(* IEC 61131-3 sources: AXOpen/src/components.robotics/ctrl/test, 2 files *)

(* ---- CylinderTests.st ---- *)
USING AXOpen.Components.Robotics;
USING AXOpen.Core;
USING AXOpen.Rtc;
USING AXOpen.Logging;

NAMESPACE Cylinder.Tests
    {S7.extern=ReadWrite}
    CLASS TestContext IMPLEMENTS AXOpen.Core.IAxoContext
        VAR
            _openCounter : ULINT;
            _closeCounter : ULINT;
        END_VAR

        METHOD PUBLIC Open : ULINT
            _openCounter := _openCounter + ULINT#1;
        END_METHOD

        METHOD PUBLIC Close : ULINT
            _closeCounter := _closeCounter + ULINT#1;
        END_METHOD

        METHOD PUBLIC CreateIdentity : ULINT
            ;
        END_METHOD

        METHOD PUBLIC OpenCycleCount : ULINT
            OpenCycleCount := _openCounter;
        END_METHOD

        METHOD PUBLIC GetRtc : AXOpen.Rtc.IAxoRtc
            ;
        END_METHOD

        METHOD PUBLIC InjectRtc
            VAR_INPUT
                Rtc : IAxoRtc;
            END_VAR

            ;
        END_METHOD

        METHOD PUBLIC GetLogger : IAxoLogger
            ;
        END_METHOD

        METHOD PUBLIC InjectLogger
            VAR_INPUT
                _logger : IAxoLogger;
            END_VAR

            ;
        END_METHOD
    END_CLASS
    {TestFixture}
    {S7.extern=ReadWrite}
    CLASS CylinderTests
        VAR
            context : TestContext;
            cylinder : ExampleCylinder;
            _homeSensor : BOOL;
            _workSensor : BOOL;
            _moveHomeSignal : BOOL;
            _moveWorkSignal : BOOL;
            _done : BOOL;
        END_VAR
        {Test}
        METHOD PUBLIC MoveHome
            WHILE _done DO
                context.Open();
                _done := Cylinder.MoveToHome.Invoke().IsDone();
                cylinder.Run(context, _homeSensor, _workSensor, _moveHomeSignal, _moveWorkSignal);
                AxUnit.Assert.Equal(_moveHomeSignal, _moveHomeSignal);
                context.Close();
            END_WHILE;

        END_METHOD
    END_CLASS
END_NAMESPACE

(* ---- RoboticsTests.st ---- *)
USING AXOpen.Components.Robotics;
USING AXOpen.Core;
USING AXOpen.Rtc;
USING AXOpen.Logging;

NAMESPACE AXOpen.Components.Robotics.Tests
    {S7.extern=ReadWrite}
    CLASS TestContext EXTENDS AXOpen.Core.Dummies.MockAxoContext
            METHOD PROTECTED OVERRIDE Main
                ;
            END_METHOD
    END_CLASS
    {TestFixture}
    {S7.extern=ReadWrite}
    CLASS RoboticsTests
        VAR
            context : TestContext;
        END_VAR
        {Test}
        METHOD PUBLIC Test1
            AxUnit.Assert.Equal(TRUE,TRUE);
        END_METHOD
    END_CLASS
END_NAMESPACE
